FUNCTION_BLOCK FB_SchmittTrigger
VAR_INPUT
    bIn: BOOL;
END_VAR
VAR_OUTPUT
    bOut: BOOL;
END_VAR
VAR
    // Number of oscillations for output switch before threshold reached
    {attribute 'hide'}
    _nLimitOscillations: INT;

    // Last input stored
    bInLast: BOOL;
    // Count of oscollations (falling / rising edge depending on bOut) while one threshold counter is active
    nOscillations: INT;
    // Time threshold to switch output after falling edge of input
    fbFallThreshold: TON;
    // Time threshold to switch output after rising edge of input
    fbRiseThreshold: TON;
END_VAR

fbFallThreshold();
fbRiseThreshold();

IF bIn <> bInLast THEN
    // Input falling edge
    IF NOT bIn THEN
        fbFallThreshold.IN := TRUE;
        fbRiseThreshold.IN := FALSE;

        // Increase oscillation counter if falling edge threashold timer has not reached tFallThreshold
        IF bOut AND NOT fbFallThreshold.Q THEN
            nOscillations := nOscillations + 1;
        END_IF

    // Input rising edge
    ELSIF bIn THEN
        fbFallThreshold.IN := FALSE;
        fbRiseThreshold.IN := TRUE;

        // Increase oscillation counter if rising edge threashold timer has not reached tRiseThreshold
        IF NOT bOut AND NOT fbRiseThreshold.Q THEN
            nOscillations := nOscillations + 1;
        END_IF
    END_IF

    // Store last input on change
    bInLast := bIn;
END_IF

// Set output bit, reset threshold timer, reset oscillation counter
IF fbFallThreshold.Q OR nLimitOscillations > 0 AND nOscillations >= nLimitOscillations AND bOut THEN
    bOut := FALSE;
    fbFallThreshold.IN := FALSE;
    nOscillations := 0;
ELSIF fbRiseThreshold.Q OR nLimitOscillations > 0 AND nOscillations >= nLimitOscillations AND NOT bOut THEN
    bOut := TRUE;
    fbRiseThreshold.IN := FALSE;
    nOscillations := 0;
END_IF

// Number of oscillations (t < threashold) required to reverse output
{attribute 'monitoring' := 'call'}
PROPERTY nLimitOscillations : INT
GET
nLimitOscillations := _nLimitOscillations;
END_GET
SET
_nLimitOscillations := nLimitOscillations;
END_SET
END_PROPERTY

// Time threshold to switch output after falling edge of input
{attribute 'monitoring' := 'call'}
PROPERTY tFallThreshold : TIME
GET
tFallThreshold := fbFallThreshold.PT;
END_GET
SET
fbFallThreshold.PT := tFallThreshold;
END_SET
END_PROPERTY

// Time threshold to switch output after rising edge of input
{attribute 'monitoring' := 'call'}
PROPERTY tRiseThreshold : TIME
GET
tRiseThreshold := fbRiseThreshold.PT;
END_GET
SET
fbRiseThreshold.PT := tRiseThreshold;
END_SET
END_PROPERTY

END_FUNCTION_BLOCK

(* stored: Version 1.1.0.1
   POU FB_SchmittTrigger: Id {5415db27-caf3-46b4-ab42-46bceaa0972b}, SpecialFunc None
   Property nLimitOscillations: Id {fed46f39-a902-4032-b67e-f208699fdedc}
   Get Get: Id {95ab3c5d-edef-4631-8b48-37459a89d486}
   Set Set: Id {684e0b90-935c-4c2f-818c-03356c664adb}
   Property tFallThreshold: Id {bcc32cd3-c8f1-4631-913d-3024989b45f9}
   Get Get: Id {9c9c8b95-49f0-4fdf-8f5e-2d8b8eeb70cc}
   Set Set: Id {dc9cb97a-faf4-4a69-8bd3-78360a0713e1}
   Property tRiseThreshold: Id {efee597b-59a7-4e11-a226-d69995658e1b}
   Get Get: Id {2534d35a-721e-41f4-bbe9-da077b4f7482}
   Set Set: Id {39139921-79cc-4cd0-a974-29a228eb2e7e} *)
